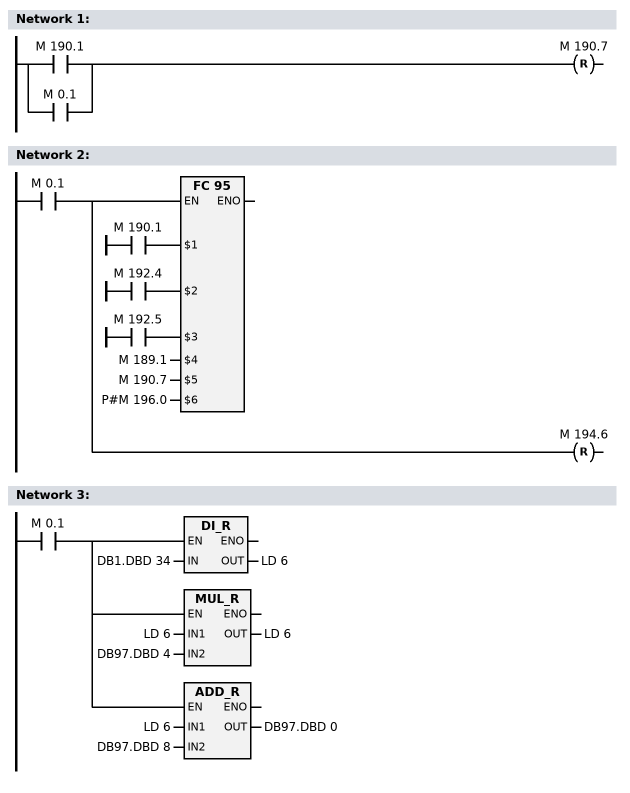
NETWORK
TITLE =
      O     M 190.1;
      O     M 0.1;
      R     M 190.7;
NETWORK
TITLE =
      A     M 0.1;
      =     L 18.0;
      A     M 190.1;
      =     L 18.1;
      BLD   103;
      A     M 192.4;
      =     L 18.2;
      BLD   103;
      A     M 192.5;
      =     L 18.3;
      BLD   103;
      A     L 18.0;
      JNB   M001;
      CALL  FC 95 (
           $1                       := L 18.1,
           $2                       := L 18.2,
           $3                       := L 18.3,
           $4                       := M 189.1,
           $5                       := M 190.7,
           $6                       := P#M 196.0);
M001: NOP   0;
      A     L 18.0;
      BLD   102;
      R     M 194.6;
NETWORK
TITLE =
      A     M 0.1;
      =     L 18.0;
      A     L 18.0;
      JNB   M002;
      L     DB1.DBD 34;
      DTR;
      T     LD 6;
M002: NOP   0;
      A     L 18.0;
      JNB   M003;
      L     LD 6;
      L     DB97.DBD 4;
      *R;
      T     LD 6;
M003: NOP   0;
      A     L 18.0;
      JNB   M004;
      L     LD 6;
      L     DB97.DBD 8;
      +R;
      T     DB97.DBD 0;
M004: NOP   0;
END_FUNCTION

FUNCTION FC 99 : VOID
AUTHOR : SKD
FAMILY : AuTPosi
NAME : CDSPL
VERSION : 0.1
BEGIN
// (block stored without names or comments; labels and parameter names are numbered)
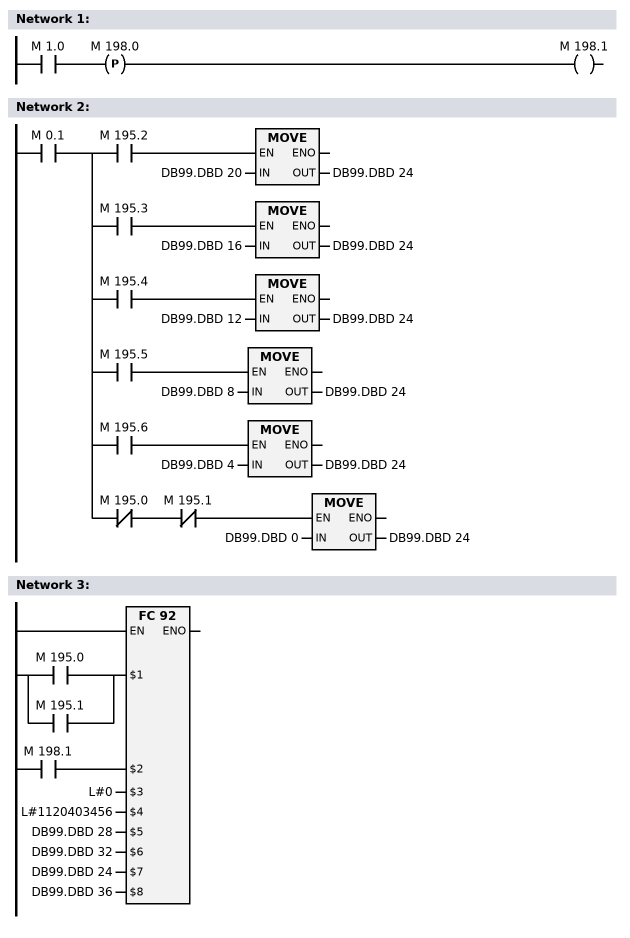
NETWORK
TITLE =
      A     M 1.0;
      FP    M 198.0;
      =     M 198.1;
NETWORK
TITLE =
      A     M 0.1;
      =     L 8.0;
      A     L 8.0;
      A     M 195.2;
      JNB   M001;
      L     DB99.DBD 20;
      T     DB99.DBD 24;
M001: NOP   0;
      A     L 8.0;
      A     M 195.3;
      JNB   M002;
      L     DB99.DBD 16;
      T     DB99.DBD 24;
M002: NOP   0;
      A     L 8.0;
      A     M 195.4;
      JNB   M003;
      L     DB99.DBD 12;
      T     DB99.DBD 24;
M003: NOP   0;
      A     L 8.0;
      A     M 195.5;
      JNB   M004;
      L     DB99.DBD 8;
      T     DB99.DBD 24;
M004: NOP   0;
      A     L 8.0;
      A     M 195.6;
      JNB   M005;
      L     DB99.DBD 4;
      T     DB99.DBD 24;
M005: NOP   0;
      A     L 8.0;
      AN    M 195.0;
      AN    M 195.1;
      JNB   M006;
      L     DB99.DBD 0;
      T     DB99.DBD 24;
M006: NOP   0;
NETWORK
TITLE =
      A(;
      O     M 195.0;
      O     M 195.1;
      );
      =     L 8.0;
      BLD   103;
      A     M 198.1;
      =     L 8.1;
      BLD   103;
      CALL  FC 92 (
           $1                       := L 8.0,
           $2                       := L 8.1,
           $3                       := L#0,
           $4                       := L#1120403456,
           $5                       := DB99.DBD 28,
           $6                       := DB99.DBD 32,
           $7                       := DB99.DBD 24,
           $8                       := DB99.DBD 36);
      NOP   0;
END_FUNCTION

FUNCTION FC 100 : VOID
AUTHOR : SKD
FAMILY : AuTiPosi
NAME : CDSPL
VERSION : 0.1
BEGIN
// (block stored without names or comments; labels and parameter names are numbered)
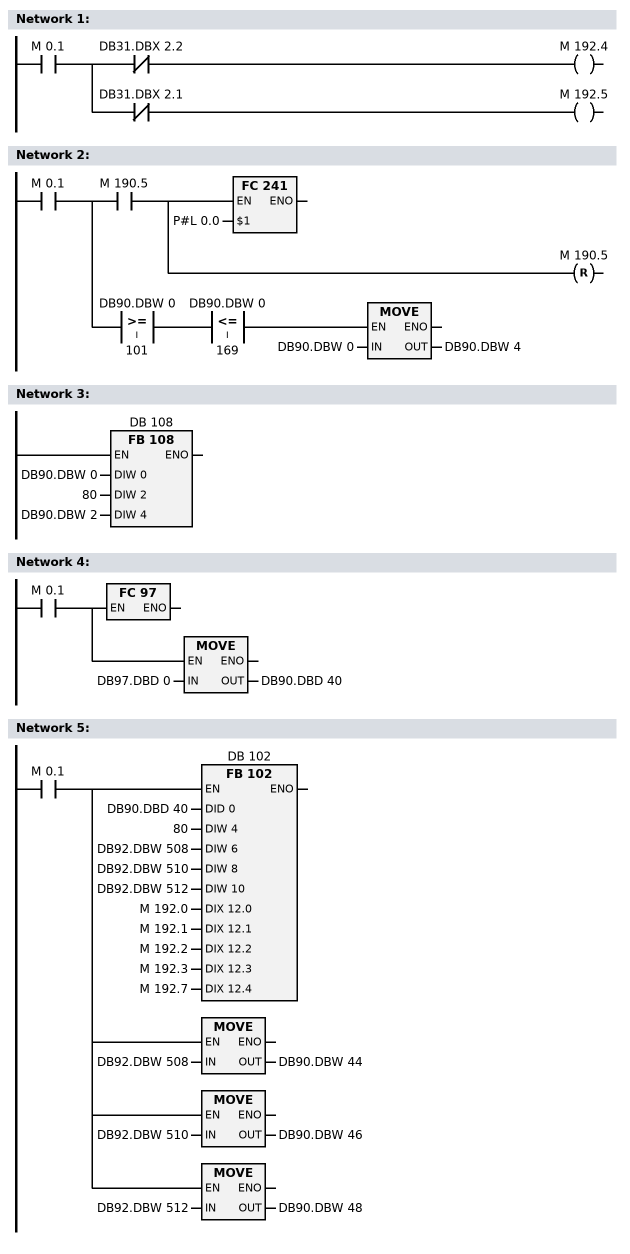
NETWORK
TITLE =
      A     M 0.1;
      =     L 6.0;
      A     L 6.0;
      AN    DB31.DBX 2.2;
      =     M 192.4;
      A     L 6.0;
      AN    DB31.DBX 2.1;
      =     M 192.5;
NETWORK
TITLE =
      A     M 0.1;
      =     L 6.0;
      A     L 6.0;
      A     M 190.5;
      =     L 6.1;
      A     L 6.1;
      JNB   M001;
      CALL  FC 241 (
           $1                       := P#L 0.0);
M001: NOP   0;
      A     L 6.1;
      BLD   102;
      R     M 190.5;
      A     L 6.0;
      A(;
      L     DB90.DBW 0;
      L     101;
      >=I;
      );
      A(;
      L     DB90.DBW 0;
      L     169;
      <=I;
      );
      JNB   M002;
      L     DB90.DBW 0;
      T     DB90.DBW 4;
M002: NOP   0;
NETWORK
TITLE =
      CALL  FB 108 , DB 108 (
           DIW 0                    := DB90.DBW 0,
           DIW 2                    := 80,
           DIW 4                    := DB90.DBW 2);
      NOP   0;
NETWORK
TITLE =
      A     M 0.1;
      =     L 6.0;
      A     L 6.0;
      JNB   M003;
      CALL  FC 97;
M003: NOP   0;
      A     L 6.0;
      JNB   M004;
      L     DB97.DBD 0;
      T     DB90.DBD 40;
M004: NOP   0;
NETWORK
TITLE =
      A     M 0.1;
      =     L 6.0;
      A     L 6.0;
      JNB   M005;
      CALL  FB 102 , DB 102 (
           DID 0                    := DB90.DBD 40,
           DIW 4                    := 80,
           DIW 6                    := DB92.DBW 508,
           DIW 8                    := DB92.DBW 510,
           DIW 10                   := DB92.DBW 512,
           DIX 12.0                 := M 192.0,
           DIX 12.1                 := M 192.1,
           DIX 12.2                 := M 192.2,
           DIX 12.3                 := M 192.3,
           DIX 12.4                 := M 192.7);
M005: NOP   0;
      A     L 6.0;
      JNB   M006;
      L     DB92.DBW 508;
      T     DB90.DBW 44;
M006: NOP   0;
      A     L 6.0;
      JNB   M007;
      L     DB92.DBW 510;
      T     DB90.DBW 46;
M007: NOP   0;
      A     L 6.0;
      JNB   M008;
      L     DB92.DBW 512;
      T     DB90.DBW 48;
M008: NOP   0;
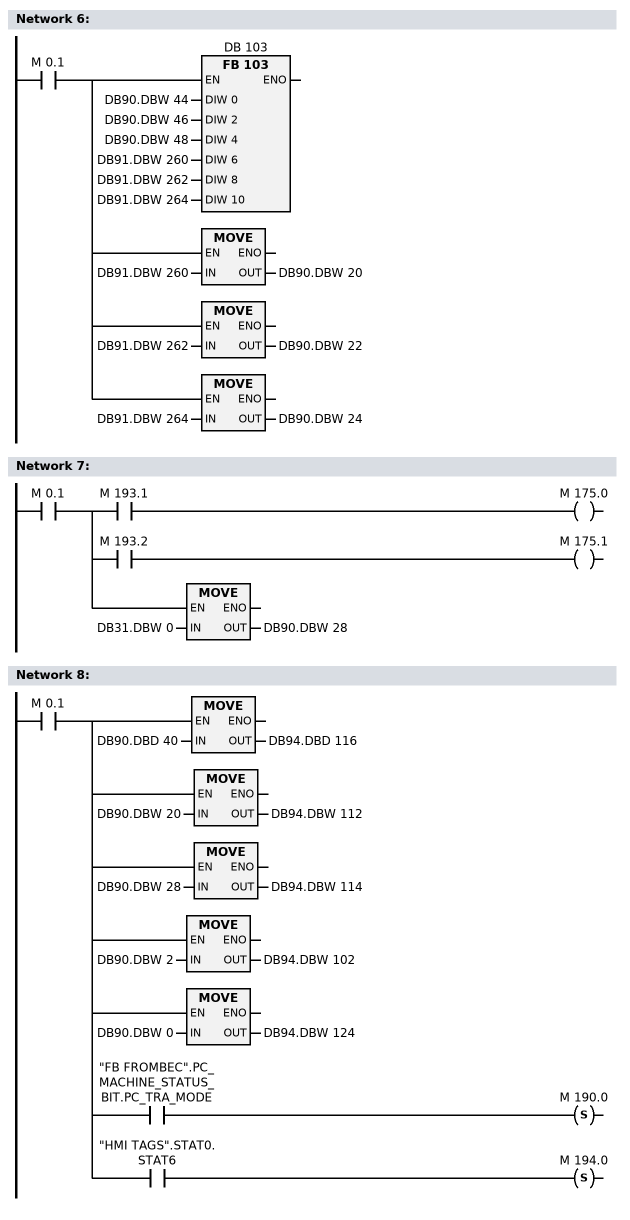
NETWORK
TITLE =
      A     M 0.1;
      =     L 6.0;
      A     L 6.0;
      JNB   M009;
      CALL  FB 103 , DB 103 (
           DIW 0                    := DB90.DBW 44,
           DIW 2                    := DB90.DBW 46,
           DIW 4                    := DB90.DBW 48,
           DIW 6                    := DB91.DBW 260,
           DIW 8                    := DB91.DBW 262,
           DIW 10                   := DB91.DBW 264);
M009: NOP   0;
      A     L 6.0;
      JNB   M010;
      L     DB91.DBW 260;
      T     DB90.DBW 20;
M010: NOP   0;
      A     L 6.0;
      JNB   M011;
      L     DB91.DBW 262;
      T     DB90.DBW 22;
M011: NOP   0;
      A     L 6.0;
      JNB   M012;
      L     DB91.DBW 264;
      T     DB90.DBW 24;
M012: NOP   0;
NETWORK
TITLE =
      A     M 0.1;
      =     L 6.0;
      A     L 6.0;
      A     M 193.1;
      =     M 175.0;
      A     L 6.0;
      A     M 193.2;
      =     M 175.1;
      A     L 6.0;
      JNB   M013;
      L     DB31.DBW 0;
      T     DB90.DBW 28;
M013: NOP   0;
NETWORK
TITLE =
      A     M 0.1;
      =     L 6.0;
      A     L 6.0;
      JNB   M014;
      L     DB90.DBD 40;
      T     DB94.DBD 116;
M014: NOP   0;
      A     L 6.0;
      JNB   M015;
      L     DB90.DBW 20;
      T     DB94.DBW 112;
M015: NOP   0;
      A     L 6.0;
      JNB   M016;
      L     DB90.DBW 28;
      T     DB94.DBW 114;
M016: NOP   0;
      A     L 6.0;
      JNB   M017;
      L     DB90.DBW 2;
      T     DB94.DBW 102;
M017: NOP   0;
      A     L 6.0;
      JNB   M018;
      L     DB90.DBW 0;
      T     DB94.DBW 124;
M018: NOP   0;
      A     L 6.0;
      A     "FB FROMBEC".PC_MACHINE_STATUS_BIT.PC_TRA_MODE;
      S     M 190.0;
      A     L 6.0;
      A     "HMI TAGS".STAT0.STAT6;
      S     M 194.0;
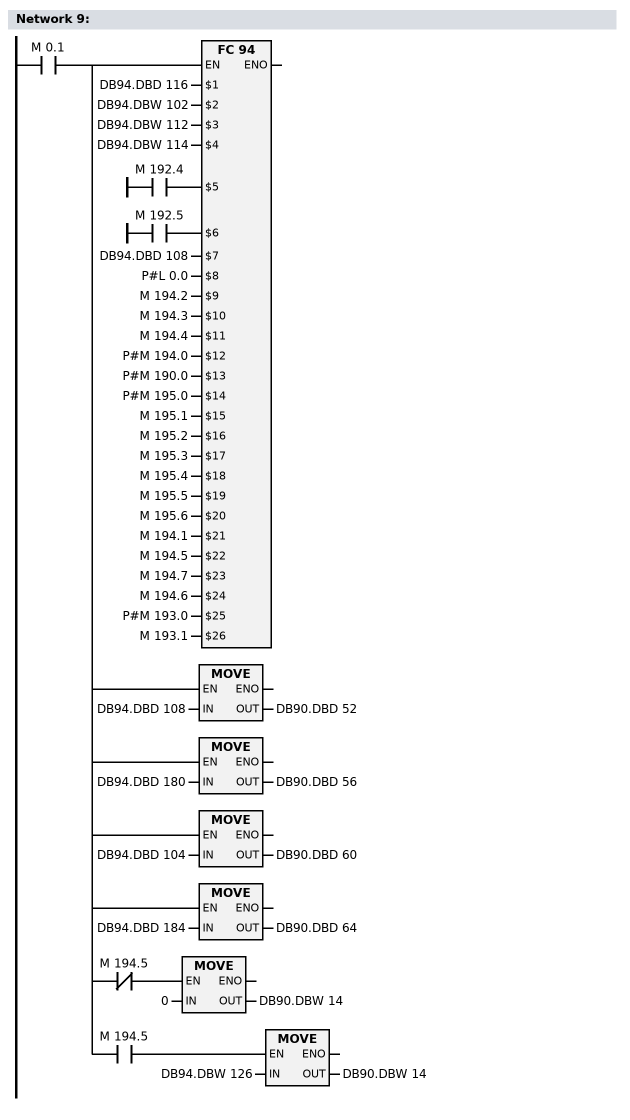
NETWORK
TITLE =
      A     M 0.1;
      =     L 6.0;
      A     M 192.4;
      =     L 6.1;
      BLD   103;
      A     M 192.5;
      =     L 6.2;
      BLD   103;
      A     L 6.0;
      JNB   M019;
      CALL  FC 94 (
           $1                       := DB94.DBD 116,
           $2                       := DB94.DBW 102,
           $3                       := DB94.DBW 112,
           $4                       := DB94.DBW 114,
           $5                       := L 6.1,
           $6                       := L 6.2,
           $7                       := DB94.DBD 108,
           $8                       := P#L 0.0,
           $9                       := M 194.2,
           $10                      := M 194.3,
           $11                      := M 194.4,
           $12                      := P#M 194.0,
           $13                      := P#M 190.0,
           $14                      := P#M 195.0,
           $15                      := M 195.1,
           $16                      := M 195.2,
           $17                      := M 195.3,
           $18                      := M 195.4,
           $19                      := M 195.5,
           $20                      := M 195.6,
           $21                      := M 194.1,
           $22                      := M 194.5,
           $23                      := M 194.7,
           $24                      := M 194.6,
           $25                      := P#M 193.0,
           $26                      := M 193.1);
M019: NOP   0;
      A     L 6.0;
      JNB   M020;
      L     DB94.DBD 108;
      T     DB90.DBD 52;
M020: NOP   0;
      A     L 6.0;
      JNB   M021;
      L     DB94.DBD 180;
      T     DB90.DBD 56;
M021: NOP   0;
      A     L 6.0;
      JNB   M022;
      L     DB94.DBD 104;
      T     DB90.DBD 60;
M022: NOP   0;
      A     L 6.0;
      JNB   M023;
      L     DB94.DBD 184;
      T     DB90.DBD 64;
M023: NOP   0;
      A     L 6.0;
      AN    M 194.5;
      JNB   M024;
      L     0;
      T     DB90.DBW 14;
M024: NOP   0;
      A     L 6.0;
      A     M 194.5;
      JNB   M025;
      L     DB94.DBW 126;
      T     DB90.DBW 14;
M025: NOP   0;
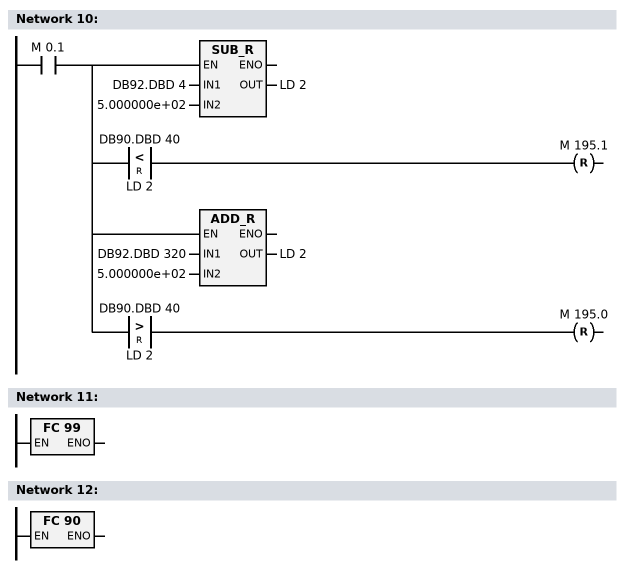
NETWORK
TITLE =
      A     M 0.1;
      =     L 6.0;
      A     L 6.0;
      JNB   M026;
      L     DB92.DBD 4;
      L     5.000000e+02;
      -R;
      T     LD 2;
M026: NOP   0;
      A     L 6.0;
      A(;
      L     DB90.DBD 40;
      L     LD 2;
      <R;
      );
      R     M 195.1;
      A     L 6.0;
      JNB   M027;
      L     DB92.DBD 320;
      L     5.000000e+02;
      +R;
      T     LD 2;
M027: NOP   0;
      A     L 6.0;
      A(;
      L     DB90.DBD 40;
      L     LD 2;
      >R;
      );
      R     M 195.0;
NETWORK
TITLE =
      CALL  FC 99;
      NOP   0;
NETWORK
TITLE =
      CALL  FC 90;
      NOP   0;
END_FUNCTION

// FC 106: know-how protected block, not included

FUNCTION FC 110 : VOID
AUTHOR : SKD
FAMILY : RaDiPosi
NAME : CDSPL
VERSION : 0.1
BEGIN
// (block stored without names or comments; labels and parameter names are numbered)
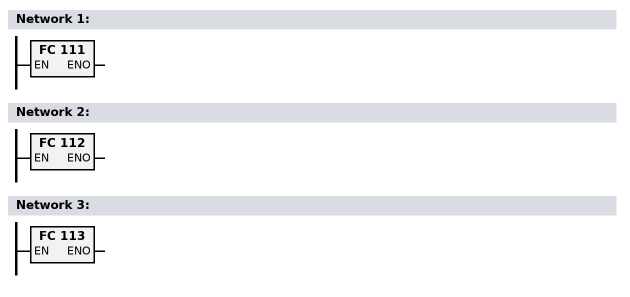
NETWORK
TITLE =
      CALL  FC 111;
      NOP   0;
NETWORK
TITLE =
      CALL  FC 112;
      NOP   0;
NETWORK
TITLE =
      CALL  FC 113;
      NOP   0;
END_FUNCTION

FUNCTION FC 111 : VOID
AUTHOR : SKD
FAMILY : AuTiPosi
NAME : CDSPL
VERSION : 0.1
BEGIN
// (block stored without names or comments; labels and parameter names are numbered)
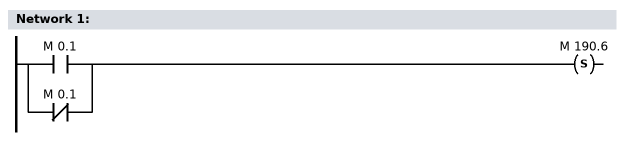
NETWORK
TITLE =
      O     M 0.1;
      ON    M 0.1;
      S     M 190.6;
END_FUNCTION

FUNCTION FC 112 : VOID
AUTHOR : SKD
FAMILY : AuTiPosi
NAME : CDSPL
VERSION : 0.1
BEGIN
// (block stored without names or comments; labels and parameter names are numbered)
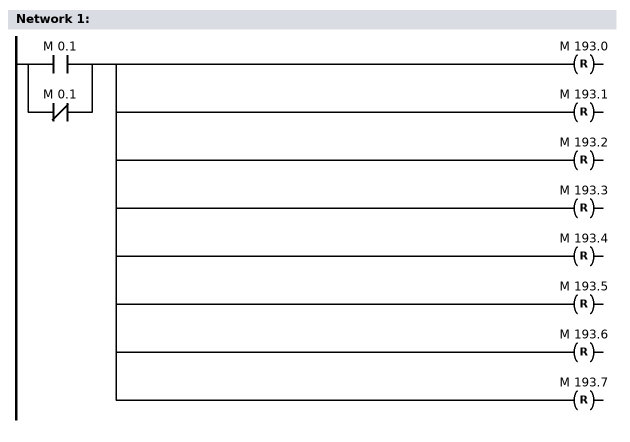
NETWORK
TITLE =
      O     M 0.1;
      ON    M 0.1;
      R     M 193.0;
      R     M 193.1;
      R     M 193.2;
      R     M 193.3;
      R     M 193.4;
      R     M 193.5;
      R     M 193.6;
      R     M 193.7;
END_FUNCTION

FUNCTION FC 113 : VOID
AUTHOR : SKD
FAMILY : AuTiPosi
NAME : CDSPL
VERSION : 0.1
BEGIN
// (block stored without names or comments; labels and parameter names are numbered)
NETWORK
TITLE =
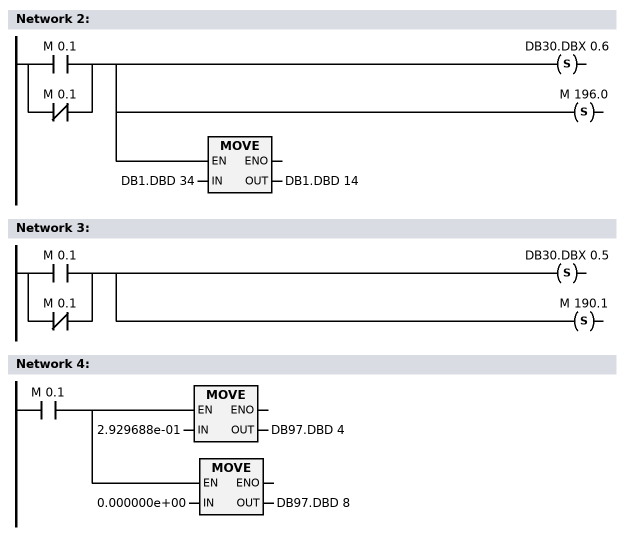
NETWORK
TITLE =
      O     M 0.1;
      ON    M 0.1;
      =     L 0.0;
      A     L 0.0;
      BLD   102;
      S     DB30.DBX 0.6;
      A     L 0.0;
      BLD   102;
      S     M 196.0;
      A     L 0.0;
      JNB   M001;
      L     DB1.DBD 34;
      T     DB1.DBD 14;
M001: NOP   0;
NETWORK
TITLE =
      O     M 0.1;
      ON    M 0.1;
      S     DB30.DBX 0.5;
      S     M 190.1;
NETWORK
TITLE =
      A     M 0.1;
      =     L 0.0;
      A     L 0.0;
      JNB   M002;
      L     2.929688e-01;
      T     DB97.DBD 4;
M002: NOP   0;
      A     L 0.0;
      JNB   M003;
      L     0.000000e+00;
      T     DB97.DBD 8;
M003: NOP   0;
END_FUNCTION

FUNCTION FC 241 : VOID
AUTHOR : SKD
FAMILY : AuTPosi
NAME : CDSPL
VERSION : 0.0
BEGIN
// (block stored without names or comments; labels and parameter names are numbered)
NETWORK
TITLE =
      SET;
      SAVE;
      =     L 0.1;
      L     DB90.DBW 0;
      L     170;
      <I;
      L     DBW 0;
      L     106;
      =     L 0.2;
      >=I;
      A     L 0.2;
      JCN   M001;
      L     DBW 4;
      L     5;
      -I;
      T     DBW 0;
      JU    M007;
M001: L     DBW 0;
      L     103;
      =     L 0.2;
      ==I;
      A     L 0.2;
      JCN   M002;
      L     168;
      T     DBW 0;
      JU    M007;
M002: L     DBW 0;
      L     104;
      =     L 0.2;
      ==I;
      A     L 0.2;
      JCN   M003;
      L     169;
      T     DBW 0;
      JU    M007;
M003: L     DBW 0;
      L     105;
      =     L 0.2;
      ==I;
      A     L 0.2;
      JCN   M004;
      L     165;
      T     DBW 0;
      JU    M007;
M004: L     DBW 0;
      L     101;
      =     L 0.2;
      ==I;
      A     L 0.2;
      JCN   M005;
      L     166;
      T     DBW 0;
      JU    M007;
M005: L     DBW 0;
      L     102;
      =     L 0.2;
      ==I;
      A     L 0.2;
      JCN   M006;
      L     167;
      T     DBW 0;
      JU    M007;
M006: L     DB90.DBW 0;
      L     101;
      >I;
      JCN   M007;
      L     169;
      T     DBW 0;
M007: L     DB90.DBW 0;
      T     #PARAM1;
      CLR;
      A     L 0.1;
      SAVE;
      BE;
END_FUNCTION

DATA_BLOCK DB 1
AUTHOR : FM
FAMILY : FM_CNT_1
NAME : CNT_CHAN
VERSION : 3.0
UDT 2
BEGIN
END_DATA_BLOCK

DATA_BLOCK "CMD TO BEC"	// DB 10
VERSION : 0.1
  STRUCT
   PC_OnBord_STATUS_BIT : STRUCT
    PC_PUSH_PERM : BOOL ;	//Pushing interlock OK
    PC_PUSH_LT_MODE : BOOL ;	//Long travel in auto or in man
    PC_TRAVEL_FWD : BOOL ;	//FWD over profibus
    PC_TRAVEL_REV : BOOL ;	//REV over profibus
    PC_TRAVEL_START : BOOL ;	//START over profibus
    PC_TRAVEL_STOP : BOOL ;	//STOP  over profibus
    GUIDE_READY : BOOL ;	//GUIDE CAR READY SIGNAL
    QLOCO_READY : BOOL ;	//QUENCHING LOCO READY SIGNAL
    PUSHER_READY : BOOL ;	//PUSHER CAR READY SIGNAL
    BATT_1_ONLINE : BOOL ;
    SpareBit_5 : BOOL ;
    SpareBit_6 : BOOL ;
    SpareBit_7 : BOOL ;
    SpareBit_8 : BOOL ;
    SpareBit_9 : BOOL ;
    SpareBit_10 : BOOL ;
    PC_SPEED_REF : INT ;	//Reserve for LT motion (spd_ref) over profibus
    SATA : ARRAY  [1 .. 7 ] OF INT ;
   END_STRUCT ;
  END_STRUCT ;	
BEGIN
END_DATA_BLOCK

DATA_BLOCK "FB FROMBEC"	// DB 11
VERSION : 0.1
  STRUCT
   PC_MACHINE_STATUS_BIT : STRUCT
    PC_PUSH_START : BOOL ;	//Pushing started
    PC_PUSH_COMPLET : BOOL ;	//Pushing completed
    PC_STATU : BOOL ;	//Status of pusher
    PC_RAM_FWD : BOOL ;	//Permissive for allowing the Ram to move fwd
    PC_STRT_LEVLING : BOOL ;	//Confirming start of leveling
    PC_STOP_LEVLING : BOOL ;	//Confirming end of leveling
    PC_PUSH_SIDE_DOOR_CL : BOOL ;	//Door open
    PC_PUSH_SIDE_DOOR_OP : BOOL ;	//Door close
    PC_DRV_STATU : BOOL ;	//Drive healthy/unhealthy
    PC_DRV_FWD : BOOL ;	//Motion towards quenching tower
    PC_DRV_REV : BOOL ;	//Motion towards coal tower
    PC_RAM_OVN_FAC_RCHD : BOOL ;	//PUSHER RAM OVEN FACE REACHED
    PC_RAM_FWD_END_RCHD : BOOL ;	//PUSHER RAM FORWARD END REACHED
    PC_TRA_MODE : BOOL ;	//PUSHER CAR TRAVEL MODE
    PC_GUIDE_CAGE_ENT : BOOL ;	//GUIDE CAGE ENTRY
    PC_HOOD_ON_CMD : BOOL ;	//HOOD SYSTEM ON COMMAND
    PC_PUSH_SPEED : REAL ;	//Pusher speed feedback
    PC_PUSH_CURRENT : INT ;	//Pusher current
    PC_RAM_POS : REAL ;	//Pusher Ram position
    PC_LEVL_CURRENT : INT ;	//LEVELER BAR DRIVE CURRENT
    SATA : ARRAY  [1 .. 2 ] OF INT ;
    PC_PUSHING_SIGNAL_START : BOOL ;
    PC_PUSHING_SIGNAL_STOP : BOOL ;
    PC_BATT_SELECT_OFFLINE : BOOL ;
    PC_BATT_SELECT_ONLINE : BOOL ;
    SPARE_1 : BOOL ;
    SPARE_2 : BOOL ;
    SPARE_3 : BOOL ;
    SPARE_4 : BOOL ;
   END_STRUCT ;
  END_STRUCT ;	
BEGIN
END_DATA_BLOCK

DATA_BLOCK DB 15
VERSION : 0.1
BEGIN
// 202 bytes; values not shown
END_DATA_BLOCK

DATA_BLOCK DB 16
VERSION : 0.1
BEGIN
// 2 bytes; values not shown
END_DATA_BLOCK

DATA_BLOCK DB 17
VERSION : 0.1
BEGIN
// 30 bytes; values not shown
END_DATA_BLOCK

DATA_BLOCK DB 18
VERSION : 0.1
BEGIN
// 34 bytes; values not shown
END_DATA_BLOCK

DATA_BLOCK DB 19
VERSION : 0.1
BEGIN
// 30 bytes; values not shown
END_DATA_BLOCK

DATA_BLOCK DB 20
VERSION : 0.1
BEGIN
// 38 bytes; values not shown
END_DATA_BLOCK

DATA_BLOCK DB 21
VERSION : 0.1
BEGIN
// 168 bytes; values not shown
END_DATA_BLOCK

DATA_BLOCK DB 22
VERSION : 0.1
BEGIN
// 66 bytes; values not shown
END_DATA_BLOCK

DATA_BLOCK DB 29
VERSION : 0.1
BEGIN
// 500 bytes; values not shown
END_DATA_BLOCK

DATA_BLOCK DB 30
VERSION : 0.1
BEGIN
// 74 bytes; values not shown
END_DATA_BLOCK

DATA_BLOCK DB 31
VERSION : 0.1
BEGIN
// 190 bytes; values not shown
END_DATA_BLOCK

DATA_BLOCK DB 32
VERSION : 0.1
BEGIN
// 48 bytes; values not shown
END_DATA_BLOCK

DATA_BLOCK "HMI TAGS"	// DB 35
VERSION : 0.1
  STRUCT
   STAT0 : STRUCT
    MODE_SEL_REQ : BOOL ;	//Mode Selection Required
    CURR_LT_MODE : BOOL ;	//Current LT Mode
    SELECT_BATTERY_1 : BOOL ;	//Battery 1 Selection Button
    SELECT_BATTERY_2 : BOOL ;	//Battery 2 Selection Button
    BATT_SELECT_OFFLINE : BOOL ;	//Battery Select Offline
    STAT6 : BOOL ;
    STAT7 : BOOL ;
    STAT8 : BOOL ;
    STAT9 : BOOL ;
    STAT10 : BOOL ;
    STAT11 : BOOL ;
    STAT12 : BOOL ;
    STAT13 : BOOL ;
    STAT14 : BOOL ;
    STAT15 : BOOL ;
    STAT16 : BOOL ;
    PUSH_STOP : BOOL ;	//Stop Pushing Button
    GC_RDY_FOR_COKE : BOOL ;	//Guide Car Ready For Coke
    QL_RDY_FOR_COKE : BOOL ;	//Quenching Loco Ready For Coke
    PUSHING_PERMISSION : BOOL ;	//Pushing Permission
    STAT21 : BOOL ;
    STAT22 : BOOL ;
    STAT23 : BOOL ;
    STAT24 : BOOL ;
    STAT25 : REAL ;
    STAT26 : REAL ;
    STAT27 : BOOL ;
    STAT28 : BOOL ;
    STAT29 : BOOL ;
    STAT30 : BOOL ;
    ALIGNMENT_BYPASS : BOOL ;	//Alignment Bypass
    STAT32 : BOOL ;
    PUSHING_PERM_ACCEPT : BOOL ;	//Pushing Permission Accept
    STAT34 : BOOL ;
    STAT35 : ARRAY  [0 .. 3 ] OF INT ;
   END_STRUCT ;
   STAT36 : STRUCT
    STAT37 : BOOL ;
    STAT38 : BOOL ;
    STAT39 : BOOL ;
    STAT40 : BOOL ;
    STAT41 : BOOL ;
    STAT42 : BOOL ;
    STAT43 : BOOL ;
    STAT44 : BOOL ;
    STAT45 : BOOL ;
    STAT46 : INT ;
    STAT47 : INT ;
    STAT48 : INT ;
    STAT49 : DINT ;
    STAT50 : ARRAY  [0 .. 8 ] OF INT ;
   END_STRUCT ;
   STAT51 : STRUCT
    STAT52 : BOOL ;
    STAT53 : BOOL ;
    STAT54 : BOOL ;
    STAT55 : BOOL ;
    STAT56 : BOOL ;
    STAT57 : BOOL ;
    STAT58 : BOOL ;
    STAT59 : BOOL ;
    STAT60 : BOOL ;
    STAT61 : BOOL ;
    STAT62 : INT ;
    STAT63 : INT ;
    STAT64 : INT ;
    STAT65 : ARRAY  [0 .. 8 ] OF INT ;
   END_STRUCT ;
   STAT66 : STRUCT
    STAT67 : BOOL ;
    STAT68 : BOOL ;
    STAT69 : BOOL ;
    STAT70 : BOOL ;
    STAT71 : BOOL ;
    STAT72 : BOOL ;
    STAT73 : BOOL ;
    STAT74 : BOOL ;
    STAT75 : BOOL ;
    STAT76 : BOOL ;
    STAT77 : INT ;
    STAT78 : INT ;
    STAT79 : INT ;
    STAT80 : ARRAY  [0 .. 8 ] OF INT ;
   END_STRUCT ;
   STAT81 : STRUCT
    STAT82 : BOOL ;
    STAT83 : BOOL ;
    STAT84 : BOOL ;
    STAT85 : BOOL ;
    STAT86 : BOOL ;
    STAT87 : BOOL ;
    STAT88 : BOOL ;
    STAT89 : BOOL ;
    STAT90 : BOOL ;
    STAT91 : BOOL ;
    STAT92 : BOOL ;
    STAT93 : INT ;
    STAT94 : INT ;
    STAT95 : INT ;
    STAT96 : REAL ;
    STAT97 : ARRAY  [0 .. 8 ] OF INT ;
   END_STRUCT ;
   STAT98 : STRUCT
    STAT99 : INT ;
    STAT100 : INT ;
    STAT101 : INT ;
    STAT102 : INT ;
    STAT103 : INT ;
    STAT104 : STRING  [1 ];
    STAT105 : STRING  [1 ];
    STAT106 : STRING  [1 ];
    STAT107 : STRING  [1 ];
    STAT108 : STRING  [1 ];
    STAT109 : STRING  [17 ];
    STAT110 : STRING  [17 ];
    STAT111 : STRING  [17 ];
    STAT112 : STRING  [17 ];
    STAT113 : STRING  [17 ];
    STAT114 : INT ;
    STAT115 : INT ;
    STAT116 : INT ;
    STAT117 : INT ;
    STAT118 : BOOL ;
    STAT119 : DINT ;
    STAT120 : INT ;
    STAT121 : INT ;
    STAT122 : STRING  [1 ];
    STAT123 : STRING  [17 ];
    STAT124 : INT ;
    STAT125 : STRING  [1 ];
    STAT126 : STRING  [17 ];
    STAT127 : BOOL ;
    STAT128 : ARRAY  [0 .. 8 ] OF DINT ;
    STAT129 : BYTE ;
   END_STRUCT ;
  END_STRUCT ;	
BEGIN
   STAT0.GC_RDY_FOR_COKE := TRUE;
   STAT0.STAT23 := TRUE;
   STAT0.STAT24 := TRUE;
   STAT0.STAT25 := 4.267091e+04;
   STAT0.STAT27 := TRUE;
   STAT0.ALIGNMENT_BYPASS := TRUE;
   STAT0.PUSHING_PERM_ACCEPT := TRUE;
   STAT36.STAT37 := TRUE;
   STAT36.STAT39 := TRUE;
   STAT36.STAT40 := TRUE;
   STAT36.STAT47 := 11;
   STAT36.STAT48 := 157;
   STAT51.STAT52 := TRUE;
   STAT51.STAT53 := TRUE;
   STAT51.STAT54 := TRUE;
   STAT51.STAT57 := TRUE;
   STAT51.STAT58 := TRUE;
   STAT51.STAT59 := TRUE;
   STAT51.STAT63 := 31;
   STAT81.STAT83 := TRUE;
   STAT81.STAT84 := TRUE;
   STAT81.STAT85 := TRUE;
   STAT81.STAT87 := TRUE;
   STAT81.STAT94 := 41;
   STAT98.STAT120 := 131;
   STAT98.STAT121 := 159;
   STAT98.STAT122 := 'C';
END_DATA_BLOCK

DATA_BLOCK DB 39
VERSION : 0.1
BEGIN
// 500 bytes; values not shown
END_DATA_BLOCK

DATA_BLOCK DB 40
VERSION : 0.1
BEGIN
// 100 bytes; values not shown
END_DATA_BLOCK

DATA_BLOCK DB 41
VERSION : 0.1
BEGIN
// 102 bytes; values not shown
END_DATA_BLOCK

DATA_BLOCK DB 50
AUTHOR : SIMATIC
FAMILY : CP341
VERSION : 0.0
FB 8
BEGIN
END_DATA_BLOCK

DATA_BLOCK DB 51
AUTHOR : SIMATIC
FAMILY : CP341
VERSION : 0.0
FB 7
BEGIN
END_DATA_BLOCK

DATA_BLOCK DB 80
AUTHOR : SIMATIC
FAMILY : CP341
VERSION : 0.0
FB 7
BEGIN
END_DATA_BLOCK

DATA_BLOCK DB 90
AUTHOR : SKD
FAMILY : AuToPosi
NAME : CDSPL
VERSION : 0.1
BEGIN
// 100 bytes; values not shown
END_DATA_BLOCK

DATA_BLOCK DB 91
AUTHOR : SKD
FAMILY : AuToPosi
NAME : CDSPL
VERSION : 0.1
BEGIN
// 310 bytes; values not shown
END_DATA_BLOCK

DATA_BLOCK DB 92
AUTHOR : SKD
FAMILY : AuToPosi
NAME : CDSPL
VERSION : 0.1
BEGIN
// 514 bytes; values not shown
END_DATA_BLOCK

DATA_BLOCK DB 94
AUTHOR : SKD
FAMILY : AuToPosi
NAME : CDSPL
VERSION : 0.1
BEGIN
// 194 bytes; values not shown
END_DATA_BLOCK

DATA_BLOCK DB 97
AUTHOR : SKD
FAMILY : AuToPosi
NAME : CDSPL
VERSION : 0.1
BEGIN
// 30 bytes; values not shown
END_DATA_BLOCK

DATA_BLOCK DB 99
AUTHOR : SKD
FAMILY : AuToPosi
NAME : CDSPL
VERSION : 0.1
BEGIN
// 40 bytes; values not shown
END_DATA_BLOCK

DATA_BLOCK DB 100
VERSION : 0.1
BEGIN
// 222 bytes; values not shown
END_DATA_BLOCK

DATA_BLOCK DB 102
VERSION : 0.0
FB 102
BEGIN
END_DATA_BLOCK

DATA_BLOCK DB 103
VERSION : 0.0
FB 103
BEGIN
END_DATA_BLOCK

DATA_BLOCK DB 108
VERSION : 0.0
FB 108
BEGIN
END_DATA_BLOCK

DATA_BLOCK DB 109
VERSION : 0.0
FB 109
BEGIN
END_DATA_BLOCK

DATA_BLOCK DB 112
VERSION : 0.0
FB 109
BEGIN
END_DATA_BLOCK

DATA_BLOCK DB 113
AUTHOR : SKD
FAMILY : AuToPosi
NAME : CDSPL
VERSION : 0.1
BEGIN
// 14 bytes; values not shown
END_DATA_BLOCK

DATA_BLOCK DB 114
VERSION : 0.0
FB 108
BEGIN
END_DATA_BLOCK

ORGANIZATION_BLOCK OB 1
AUTHOR : SKD
NAME : CDSPL
VERSION : 0.1
BEGIN
// (block stored without names or comments; labels and parameter names are numbered)
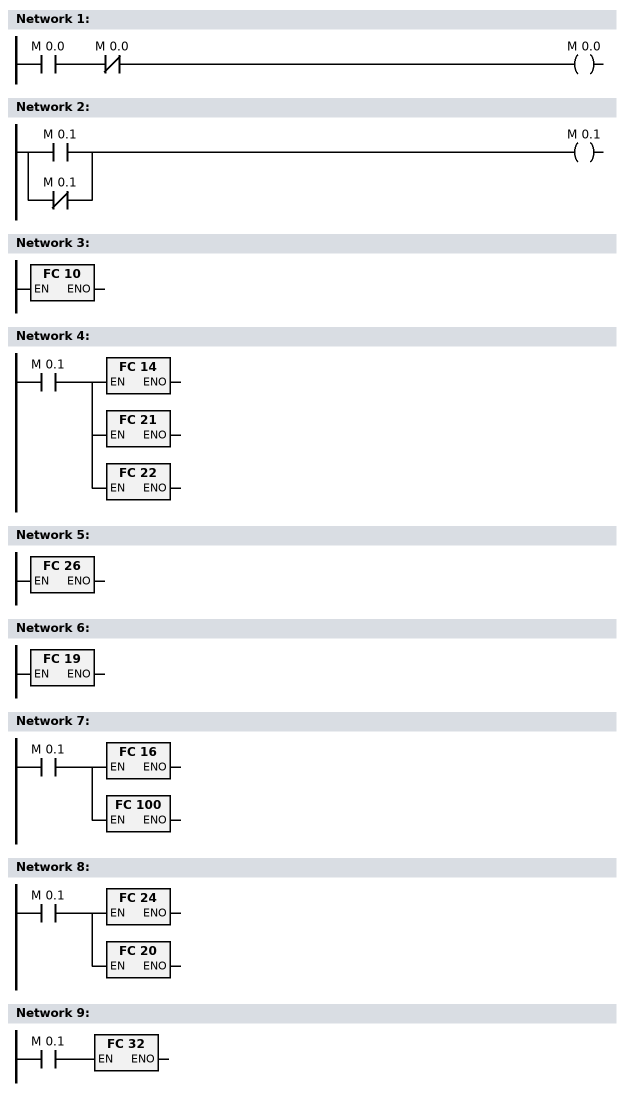
NETWORK
TITLE =
      A     M 0.0;
      AN    M 0.0;
      =     M 0.0;
NETWORK
TITLE =
      O     M 0.1;
      ON    M 0.1;
      =     M 0.1;
NETWORK
TITLE =
      CALL  FC 10;
      NOP   0;
NETWORK
TITLE =
      A     M 0.1;
      =     L 20.0;
      A     L 20.0;
      JNB   M001;
      CALL  FC 14;
M001: NOP   0;
      A     L 20.0;
      JNB   M002;
      CALL  FC 21;
M002: NOP   0;
      A     L 20.0;
      JNB   M003;
      CALL  FC 22;
M003: NOP   0;
NETWORK
TITLE =
      CALL  FC 26;
      NOP   0;
NETWORK
TITLE =
      CALL  FC 19;
      NOP   0;
NETWORK
TITLE =
      A     M 0.1;
      =     L 20.0;
      A     L 20.0;
      JNB   M004;
      CALL  FC 16;
M004: NOP   0;
      A     L 20.0;
      JNB   M005;
      CALL  FC 100;
M005: NOP   0;
NETWORK
TITLE =
      A     M 0.1;
      =     L 20.0;
      A     L 20.0;
      JNB   M006;
      CALL  FC 24;
M006: NOP   0;
      A     L 20.0;
      JNB   M007;
      CALL  FC 20;
M007: NOP   0;
NETWORK
TITLE =
      A     M 0.1;
      JNB   M008;
      CALL  FC 32;
M008: NOP   0;
END_ORGANIZATION_BLOCK

ORGANIZATION_BLOCK OB 82
VERSION : 0.1
BEGIN
// (block stored without names or comments; labels and parameter names are numbered)
NETWORK
TITLE =
      SET;
      S     DB30.DBX 54.1;
      S     DB30.DBX 54.0;
      CALL  FC 4 (
           $1                       := 1,
           $2                       := DB30.DBW 72,
           $3                       := DB30.DBX 54.0);
END_ORGANIZATION_BLOCK

ORGANIZATION_BLOCK OB 86
VERSION : 0.1
BEGIN
// (block stored without names or comments; labels and parameter names are numbered)
NETWORK
TITLE =
END_ORGANIZATION_BLOCK

ORGANIZATION_BLOCK OB 100
VERSION : 0.1
BEGIN
// (block stored without names or comments; labels and parameter names are numbered)
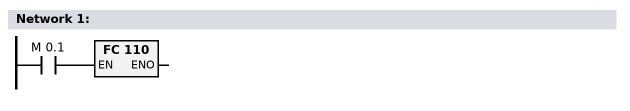
NETWORK
TITLE =
      A     M 0.1;
      JNB   M001;
      CALL  FC 110;
M001: NOP   0;
END_ORGANIZATION_BLOCK

ORGANIZATION_BLOCK OB 121
VERSION : 0.1
BEGIN
// (block stored without names or comments; labels and parameter names are numbered)
NETWORK
TITLE =
END_ORGANIZATION_BLOCK

ORGANIZATION_BLOCK OB 122
VERSION : 0.1
BEGIN
// (block stored without names or comments; labels and parameter names are numbered)
NETWORK
TITLE =
END_ORGANIZATION_BLOCK
